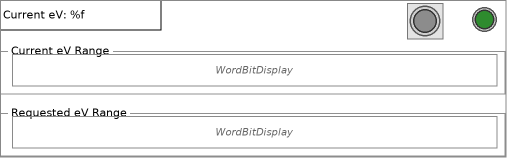
VISUALIZATION PhotonEnergyWatcher  // 507x158
VAR_IN_OUT
	Watcher	:	FB_PhotonEnergyWatcher;
END_VAR
    GroupBox (0,43 505x51), "Current eV Range"
        Frame (12,11 485x32)
            shows WordBitDisplay(nVal := Watcher.i_stCurrentBeamParams.neVRange)
    Rectangle (0,0 161x30), "Current eV: %f", text variable: Watcher.i_stCurrentBeamParams.reV
    GroupBox (0,105 505x51), "Requested eV Range"
        Frame (12,11 485x32)
            shows WordBitDisplay(nVal := Watcher.i_stRequestedBeamParams.neVRange)
    Lamp1 (470,2 29x35), variable: Watcher.fbFF.bsFF.Q1, style: Lamp-Lamp1-Green
    PushSwitch (407,1 36x40), variable: Watcher.i_xReset, behaviour: TAP, style: Switch-PushSwitch-Gray
END_VISUALIZATION

(* stored: Version 1.1.0.1, ProductVersion 3.1.4024.0
   Visu PhotonEnergyWatcher: Id {48fceb58-0778-0e47-2f10-bb988f882783} *)
